(* IEC 61131-3 sources: F100R_S278_Temperville/MyController.device.xml.v3^/Plc Logic.plclogic.xml.v3^/Application.application.xml.v3^/10_EntradasSaidas, 3 files *)

(* ---- A_Principal_IO.prg.st ---- *)
PROGRAM A_Principal_IO

IF NOT xTesteEntradaSaidas THEN
	B_EspelhoEntradas();
	C_EspelhoSaida();
END_IF

(* ---- B_EspelhoEntradas.prg.st ---- *)
PROGRAM B_EspelhoEntradas
VAR

END_VAR

//TM262L10MESE8T - 0.1

ImgTesteEntradas[1]:=   xChCircuitoEmergenciaCC	:= xM0_1_DI0;//xChCircuitoEmergenciaCC
ImgTesteEntradas[2]:=   xChHabDesabCircuitoCC := xM0_1_DI1;//Reserva
ImgTesteEntradas[3]:=   xSaidaNobreakOk:= 	xM0_1_DI2;//xSaidaNobreakOk
ImgTesteEntradas[4]:=	xReleSeguranca:=	xM0_1_DI3;//xReleSeguranca

xInvVentilador01Habilitado:=true;//xM0_1_DI1;

//TM3XHSC202 - 0.2
ImgTesteEntradas[5]:=	xM0_2_DI0;// ENCODER
ImgTesteEntradas[6]:=	xM0_2_DI1;// ENCODER
ImgTesteEntradas[7]:=	xM0_2_DI2;// ENCODER
ImgTesteEntradas[8]:=	xM0_2_DI3;// ENCODER
ImgTesteEntradas[9]:=	xM0_2_DI4;// ENCODER
ImgTesteEntradas[10]:=	xM0_2_DI5;// ENCODER
ImgTesteEntradas[11]:=	xM0_2_DI6;// ENCODER
ImgTesteEntradas[12]:=	xM0_2_DI7;// ENCODER
ImgTesteEntradas[13]:=	xM0_2_DI8;// ENCODER
ImgTesteEntradas[14]:=	xM0_2_DI9;// ENCODER

//TM3XHSC202 - 0.3
ImgTesteEntradas[15]:=	xM0_3_DI0;// ENCODER
ImgTesteEntradas[16]:=	xM0_3_DI1;// ENCODER
ImgTesteEntradas[17]:=	xM0_3_DI2;// ENCODER
ImgTesteEntradas[18]:=	xM0_3_DI3;// ENCODER
ImgTesteEntradas[19]:=	xM0_3_DI4;// ENCODER
ImgTesteEntradas[20]:=	xM0_3_DI5;// ENCODER
ImgTesteEntradas[21]:=	xM0_3_DI6;// ENCODER
ImgTesteEntradas[22]:=	xM0_3_DI7;// ENCODER
ImgTesteEntradas[23]:=	xM0_3_DI8;// ENCODER
ImgTesteEntradas[24]:=	xM0_3_DI9;// ENCODER

//TM3DI32K - 0.4
ImgTesteEntradas[25]:= 	xChAvancaMesaEntrada	:= xM0_4_DI0;	//xChAvancaMesaEntrada
ImgTesteEntradas[26]:= 	xChRecuaMesaEntrada		:= xM0_4_DI1;	//xChRecuaMesaEntrada
ImgTesteEntradas[27]:= 	xSensorEntrada01		:= xM0_4_DI2;	//xSensorEntrada01
ImgTesteEntradas[28]:= 	xSensorEntrada02		:= xM0_4_DI3;	//xSensorEntrada02
ImgTesteEntradas[29]:= 	xSensorEntrada03		:= xM0_4_DI4;	//xSensorEntrada03
ImgTesteEntradas[30]:= 	xSensorEntrada04		:= xM0_4_DI5;	//xSensorEntrada04
ImgTesteEntradas[31]:= 	xSensorEntrada05		:= xM0_4_DI6;	//xSensorEntrada05
ImgTesteEntradas[32]:= 	xSensorEntrada06		:= xM0_4_DI7;  //xSensorEntrada06
ImgTesteEntradas[33]:= 	xSensorEntrada07		:= xM0_4_DI8;  //xSensorEntrada07
ImgTesteEntradas[34]:= 	xSensorEntrada08		:= xM0_4_DI9;  //xSensorEntrada08
ImgTesteEntradas[35]:= 	xBtGradeEntrada			:= xM0_4_DI10; //xBtGradeEntrada
ImgTesteEntradas[36]:= 	xBtHabilitaCarregamento	:= xM0_4_DI11; //xBtHabilitaCarregamento
ImgTesteEntradas[37]:= 	xBt02Emergencia			:= xM0_4_DI12; //xBt02Emergencia Mesa Entrada
ImgTesteEntradas[38]:= 	xSensorPortaEntrada		:= xM0_4_DI13; //xSensorPortaEntrada
ImgTesteEntradas[39]:= 	xSensorPortaSaida		:=	xM0_4_DI14; //xSensorPortaSaida
ImgTesteEntradas[40]:= 	xM0_4_DI15; //xSensorAbertoForno
ImgTesteEntradas[41]:=	xM0_4_DI16; //xSensorFechadoForno
ImgTesteEntradas[42]:=	xSensorAbertoResfriadorSup02:= xM0_4_DI17; //xSensorAbertoResfriadorSup02
ImgTesteEntradas[43]:=	xSensorFechadoResfriadorSup02:= xM0_4_DI18; //xSensorFechadoResfriadorSup02
ImgTesteEntradas[44]:=	xFcMaximoSegResfriadorSup02:= xM0_4_DI19; //xFcMaximoSegResfriadorSup02
ImgTesteEntradas[45]:=	xFcMinimoSegResfriadorSup02:= xM0_4_DI20; //xFcMinimoSegResfriadorSup02
ImgTesteEntradas[46]:=	xChAbreDuctosResfriadorSup02:= xM0_4_DI21; //xChAbreDuctosResfriadorSup02
ImgTesteEntradas[47]:=	xBt03Emergencia			:= xM0_4_DI22; //xBt03Emergencia Mesa Resfriador
ImgTesteEntradas[48]:=	xSensorDesligaMesaSaida	:= xM0_4_DI23; //xSensorDesligaMesaSaida
ImgTesteEntradas[49]:=	xSensorGradeSaidaUp		:= xM0_4_DI24; //xSensorGradeSaidaUp
ImgTesteEntradas[50]:=	xBtGradeSaida			:=	xM0_4_DI25;  //	xBtGradeSaida
ImgTesteEntradas[51]:=	xChAvancaMesaSaida		:= xM0_4_DI26; //xChAvancaMesaSaida
ImgTesteEntradas[52]:=	xChRecuaMesaSaida		:=	xM0_4_DI27; //xChRecuaMesaSaida
ImgTesteEntradas[53]:=	xBt04Emergencia			:= xM0_4_DI28; //xBt04Emergencia Mesa Saída
ImgTesteEntradas[54]:=	xSensorPositivoGuilhotina02:= xM0_4_DI29; //xSensorPositivoGuilhotina02
ImgTesteEntradas[55]:=	xSensorNegativoGuilhotina02:=xM0_4_DI30; //xSensorNegativoGuilhotina02
ImgTesteEntradas[56]:=	xSensorZeroGuilhotina02	:= xM0_4_DI31; //xSensorZeroGuilhotina02

//TM3DI32K - 3.1
ImgTesteEntradas[57]:= 	xChAutomaticoManual:= xM3_1_DI0;   //xChAutomaticoManual
ImgTesteEntradas[58]:= xBt01CalaAlarme:= xM3_1_DI1;   //xBt01CalaAlarme Mesa Controle
ImgTesteEntradas[59]:= xBt01Emergencia:= xM3_1_DI2;   //xBt01Emergencia Mesa Controle
ImgTesteEntradas[60]:= xPressaoBaixaMediaRede:= xM3_1_DI3;   //xPressaoBaixaMediaRede
ImgTesteEntradas[61]:= xPressaoMediaAltaRede:=	xM3_1_DI4;   //xPressaoMediaAltaRede
ImgTesteEntradas[62]:= xKaMotorOscilaResfr02Sup:= xM3_1_DI5;   //oscilantes
ImgTesteEntradas[63]:= xKaMotorOscilaResfr02Inf:= xM3_1_DI6;   //oscilantes
ImgTesteEntradas[64]:= xSensorOscilaResfr02Sup:= xM3_1_DI7;   //oscilantes
ImgTesteEntradas[65]:= xSensorOscilaResfr02Inf:= xM3_1_DI8;   //oscilantes
ImgTesteEntradas[66]:= xRetornoSsr01ConveccaoEnt:=	xM3_1_DI9;   //xRetornoSsr01ConveccaoEnt
ImgTesteEntradas[67]:= xRetornoSsr02ConveccaoEnt:=	xM3_1_DI10;  //xRetornoSsr02ConveccaoEnt
ImgTesteEntradas[68]:= xRetornoSsr03ConveccaoEnt:=	xM3_1_DI11;  //xRetornoSsr03ConveccaoEnt
ImgTesteEntradas[69]:= xRetornoSsrInferior[1]:= xM3_1_DI12;  //Retorno Circuito Resist Inf 01
ImgTesteEntradas[70]:= xRetornoSsrInferior[2]:= xM3_1_DI13;  //Retorno Circuito Resist Inf 02
ImgTesteEntradas[71]:= xRetornoSsrInferior[3]:= xM3_1_DI14;  //Retorno Circuito Resist Inf 03
ImgTesteEntradas[72]:= xRetornoSsrInferior[4]:= xM3_1_DI15;  //Retorno Circuito Resist Inf 04

//TM3DI32K - 3.2
ImgTesteEntradas[73]:= xRetornoSsrInferior[5]:= xM3_2_DI0;   //Retorno Circuito Resist Inf 05
ImgTesteEntradas[74]:= xRetornoSsrInferior[6]:= xM3_2_DI1;   //Retorno Circuito Resist Inf 06
ImgTesteEntradas[75]:= xRetornoSsrInferior[7]:= xM3_2_DI2;   //Retorno Circuito Resist Inf 07
ImgTesteEntradas[76]:= xRetornoSsrInferior[8]:= xM3_2_DI3;   //Retorno Circuito Resist Inf 08
ImgTesteEntradas[77]:= xRetornoSsrInferior[9]:= xM3_2_DI4;   //Retorno Circuito Resist Inf 09
ImgTesteEntradas[78]:= xRetornoSsrInferior[10]:= xM3_2_DI5;   //Retorno Circuito Resist Inf 10
ImgTesteEntradas[79]:= xRetornoSsrInferior[11]:= xM3_2_DI6;   //Retorno Circuito Resist Inf 11
ImgTesteEntradas[80]:= xRetornoSsrInferior[12]:= xM3_2_DI7;   //Retorno Circuito Resist Inf 12
ImgTesteEntradas[81]:= xRetornoSsrInferior[13]:= xM3_2_DI8;   //Retorno Circuito Resist Inf 13
ImgTesteEntradas[82]:= xRetornoSsrInferior[14]:= xM3_2_DI9;   //Retorno Circuito Resist Inf 14
ImgTesteEntradas[83]:= xRetornoSsrInferior[15]:= xM3_2_DI10;  //Retorno Circuito Resist Inf 15
ImgTesteEntradas[84]:= xRetornoSsrInferior[16]:= xM3_2_DI11;  //Retorno Circuito Resist Inf 16
ImgTesteEntradas[85]:= xRetornoSsrInferior[17]:= xM3_2_DI12;  //Retorno Circuito Resist Inf 17
ImgTesteEntradas[86]:= xRetornoSsrInferior[18]:= xM3_2_DI13;  //Retorno Circuito Resist Inf 18
ImgTesteEntradas[87]:= xRetornoSsrInferior[19]:= xM3_2_DI14;  //Retorno Circuito Resist Inf 19
ImgTesteEntradas[88]:= xRetornoSsrInferior[20]:= xM3_2_DI15;  //Retorno Circuito Resist Inf 20
ImgTesteEntradas[89]:= xRetornoSsrInferior[21]:= xM3_2_DI16;  //Retorno Circuito Resist Inf 21
ImgTesteEntradas[90]:= xRetornoSsrInferior[22]:= xM3_2_DI17;  //Retorno Circuito Resist Inf 22
ImgTesteEntradas[91]:= xRetornoSsrInferior[23]:= xM3_2_DI18;  //Retorno Circuito Resist Inf 23
ImgTesteEntradas[92]:= xRetornoSsrInferior[24]:= xM3_2_DI19;  //Retorno Circuito Resist Inf 24
ImgTesteEntradas[93]:= xRetornoSsrInferior[25]:= xM3_2_DI20;  //Retorno Circuito Resist Inf 25
ImgTesteEntradas[94]:= xRetornoSsrInferior[26]:= xM3_2_DI21;  //Retorno Circuito Resist Inf 26
ImgTesteEntradas[95]:= xRetornoSsrInferior[27]:= xM3_2_DI22;  //Retorno Circuito Resist Inf 27
ImgTesteEntradas[96]:= xRetornoSsrInferior[28]:= xM3_2_DI23;  //Retorno Circuito Resist Inf 28
ImgTesteEntradas[97]:= xRetornoSsrInferior[29]:= xM3_2_DI24;  //Retorno Circuito Resist Inf 29
ImgTesteEntradas[98]:= xRetornoSsrInferior[30]:= xM3_2_DI25;  //Retorno Circuito Resist Inf 30
ImgTesteEntradas[99]:= xRetornoSsrInferior[31]:= xM3_2_DI26;  //Retorno Circuito Resist Inf 31
ImgTesteEntradas[100]:= xRetornoSsrInferior[32]:= xM3_2_DI27;  //Retorno Circuito Resist Inf 32
ImgTesteEntradas[101]:=	xRetornoSsrInferior[33]:= xM3_2_DI28;  //Retorno Circuito Resist Inf 33
ImgTesteEntradas[102]:=	xRetornoSsrInferior[34]:= xM3_2_DI29;  //Retorno Circuito Resist Inf 34
ImgTesteEntradas[103]:=	xRetornoSsrInferior[35]:= xM3_2_DI30;  //Retorno Circuito Resist Inf 35
ImgTesteEntradas[104]:=	xRetornoSsrInferior[36]:= xM3_2_DI31;  //Retorno Circuito Resist Inf 36

//TM3DI32K - 4.1
ImgTesteEntradas[105]:=	xRetornoSsrInferior[37]:= xM4_1_DI0;   //Retorno Circuito Resist Inf 37
ImgTesteEntradas[106]:=	xRetornoSsrInferior[38]:= xM4_1_DI1;   //Retorno Circuito Resist Inf 38
ImgTesteEntradas[107]:=	xRetornoSsrInferior[39]:= xM4_1_DI2;   //Retorno Circuito Resist Inf 39
ImgTesteEntradas[108]:=	xRetornoSsrInferior[40]:= xM4_1_DI3;   //Retorno Circuito Resist Inf 40
ImgTesteEntradas[109]:=	xRetornoSsrInferior[41]:= xM4_1_DI4;   //Retorno Circuito Resist Inf 41
ImgTesteEntradas[110]:=	xRetornoSsrInferior[42]:= xM4_1_DI5;   //Retorno Circuito Resist Inf 42
ImgTesteEntradas[111]:=	xRetornoSsrInferior[43]:= xM4_1_DI6;   //Retorno Circuito Resist Inf 43
ImgTesteEntradas[112]:=	xRetornoSsrInferior[44]:= xM4_1_DI7;   //Retorno Circuito Resist Inf 44
ImgTesteEntradas[113]:=	xRetornoSsrInferior[45]:= xM4_1_DI8;   //Retorno Circuito Resist Inf 45
ImgTesteEntradas[114]:=	xRetornoSsrInferior[46]:= xM4_1_DI9;   //Retorno Circuito Resist Inf 46
ImgTesteEntradas[115]:=	xRetornoSsrInferior[47]:= xM4_1_DI10;  //Retorno Circuito Resist Inf 47
ImgTesteEntradas[116]:=	xRetornoSsrInferior[48]:= xM4_1_DI11;  //Retorno Circuito Resist Inf 48
ImgTesteEntradas[117]:=	xRetornoSsrInferior[49]:= xM4_1_DI12;  //Retorno Circuito Resist Inf 49
ImgTesteEntradas[118]:= xRetornoSsrInferior[50]:= xM4_1_DI13;  //Retorno Circuito Resist Inf 50
ImgTesteEntradas[119]:= xRetornoSsrSuperior[1]:= xM4_1_DI14;  //Retorno Circuito Resist Sup 01 - 51
ImgTesteEntradas[120]:= xRetornoSsrSuperior[2]:= xM4_1_DI15;  //Retorno Circuito Resist Sup 02 - 52
ImgTesteEntradas[121]:= xRetornoSsrSuperior[3]:= xM4_1_DI16;  //Retorno Circuito Resist Sup 03 - 53
ImgTesteEntradas[122]:= xRetornoSsrSuperior[4]:= xM4_1_DI17;  //Retorno Circuito Resist Sup 04 - 54
ImgTesteEntradas[123]:= xRetornoSsrSuperior[5]:= xM4_1_DI18;  //Retorno Circuito Resist Sup 05 - 55
ImgTesteEntradas[124]:= xRetornoSsrSuperior[6]:= xM4_1_DI19;  //Retorno Circuito Resist Sup 06 - 56
ImgTesteEntradas[125]:= xRetornoSsrSuperior[7]:= xM4_1_DI20;  //Retorno Circuito Resist Sup 07 - 57
ImgTesteEntradas[126]:= xRetornoSsrSuperior[8]:= xM4_1_DI21;  //Retorno Circuito Resist Sup 08 - 58
ImgTesteEntradas[127]:= xRetornoSsrSuperior[9]:= xM4_1_DI22;  //Retorno Circuito Resist Sup 09 - 59
ImgTesteEntradas[128]:= xRetornoSsrSuperior[10]:= xM4_1_DI23;  //Retorno Circuito Resist Sup 10 - 60
ImgTesteEntradas[129]:= xRetornoSsrSuperior[11]:= xM4_1_DI24;  //Retorno Circuito Resist Sup 11 - 61
ImgTesteEntradas[130]:= xRetornoSsrSuperior[12]:= xM4_1_DI25;  //Retorno Circuito Resist Sup 12 - 62
ImgTesteEntradas[131]:= xRetornoSsrSuperior[13]:= xM4_1_DI26;  //Retorno Circuito Resist Sup 13 - 63
ImgTesteEntradas[132]:= xRetornoSsrSuperior[14]:= xM4_1_DI27;  //Retorno Circuito Resist Sup 14 - 64
ImgTesteEntradas[133]:=	xRetornoSsrSuperior[15]:= xM4_1_DI28;  //Retorno Circuito Resist Sup 15 - 65
ImgTesteEntradas[134]:=	xRetornoSsrSuperior[16]:= xM4_1_DI29;  //Retorno Circuito Resist Sup 16 - 66
ImgTesteEntradas[135]:=	xRetornoSsrSuperior[17]:= xM4_1_DI30;  //Retorno Circuito Resist Sup 17 - 67
ImgTesteEntradas[136]:=	xRetornoSsrSuperior[18]:= xM4_1_DI31;  //Retorno Circuito Resist Sup 18 - 68

//TM3DI32K - 4.2
ImgTesteEntradas[137]:= xRetornoSsrSuperior[19]:= xM4_2_DI0;   //Retorno Circuito Resist Sup 19	- 69
ImgTesteEntradas[138]:= xRetornoSsrSuperior[20]:= xM4_2_DI1;   //Retorno Circuito Resist Sup 20	- 70
ImgTesteEntradas[139]:= xRetornoSsrSuperior[21]:= xM4_2_DI2;   //Retorno Circuito Resist Sup 21	- 71
ImgTesteEntradas[140]:= xRetornoSsrSuperior[22]:= xM4_2_DI3;   //Retorno Circuito Resist Sup 22	- 72
ImgTesteEntradas[141]:= xRetornoSsrSuperior[23]:= xM4_2_DI4;   //Retorno Circuito Resist Sup 23	- 73
ImgTesteEntradas[142]:= xRetornoSsrSuperior[24]:= xM4_2_DI5;   //Retorno Circuito Resist Sup 24	- 74
ImgTesteEntradas[143]:= xRetornoSsrSuperior[25]:= xM4_2_DI6;   //Retorno Circuito Resist Sup 25	- 75
ImgTesteEntradas[144]:= xRetornoSsrSuperior[26]:= xM4_2_DI7;   //Retorno Circuito Resist Sup 26	- 76
ImgTesteEntradas[145]:= xRetornoSsrSuperior[27]:= xM4_2_DI8;   //Retorno Circuito Resist Sup 27	- 77
ImgTesteEntradas[146]:= xRetornoSsrSuperior[28]:= xM4_2_DI9;   //Retorno Circuito Resist Sup 28 - 78
ImgTesteEntradas[147]:= xRetornoSsrSuperior[29]:= xM4_2_DI10;  //Retorno Circuito Resist Sup 29	- 79
ImgTesteEntradas[148]:= xRetornoSsrSuperior[30]:= xM4_2_DI11;  //Retorno Circuito Resist Sup 30	- 80
ImgTesteEntradas[149]:= xRetornoSsrSuperior[31]:= xM4_2_DI12;  //Retorno Circuito Resist Sup 31	- 81
ImgTesteEntradas[150]:= xRetornoSsrSuperior[32]:= xM4_2_DI13;  //Retorno Circuito Resist Sup 32	- 82
ImgTesteEntradas[151]:= xRetornoSsrSuperior[33]:= xM4_2_DI14;  //Retorno Circuito Resist Sup 33 - 83
ImgTesteEntradas[152]:= xRetornoSsrSuperior[34]:= xM4_2_DI15;  //Retorno Circuito Resist Sup 34 - 84
ImgTesteEntradas[153]:= xRetornoSsrSuperior[35]:= xM4_2_DI16;  //Retorno Circuito Resist Sup 35 - 85
ImgTesteEntradas[154]:= xRetornoSsrSuperior[36]:= xM4_2_DI17;  //Retorno Circuito Resist Sup 36 - 86
ImgTesteEntradas[155]:= xRetornoSsrSuperior[37]:= xM4_2_DI18;  //Retorno Circuito Resist Sup 37	- 87
ImgTesteEntradas[156]:= xRetornoSsrSuperior[38]:= xM4_2_DI19;  //Retorno Circuito Resist Sup 38	- 88
ImgTesteEntradas[157]:= xRetornoSsrSuperior[39]:= xM4_2_DI20;  //Retorno Circuito Resist Sup 39 - 89
ImgTesteEntradas[158]:= xRetornoSsrSuperior[40]:= xM4_2_DI21;  //Retorno Circuito Resist Sup 40	- 90
ImgTesteEntradas[159]:= xRetornoSsrSuperior[41]:= xM4_2_DI22;  //Retorno Circuito Resist Sup 41 - 91
ImgTesteEntradas[160]:= xRetornoSsrSuperior[42]:= xM4_2_DI23;  //Retorno Circuito Resist Sup 42 - 92
ImgTesteEntradas[161]:= xRetornoSsrSuperior[43]:= xM4_2_DI24;  //Retorno Circuito Resist Sup 43 - 93
ImgTesteEntradas[162]:= xRetornoSsrSuperior[44]:= xM4_2_DI25;  //Retorno Circuito Resist Sup 44 - 94
ImgTesteEntradas[163]:= xRetornoSsrSuperior[45]:= xM4_2_DI26;  //Retorno Circuito Resist Sup 45 - 95
ImgTesteEntradas[164]:= xRetornoSsrSuperior[46]:= xM4_2_DI27;  //Retorno Circuito Resist Sup 46 - 96
ImgTesteEntradas[165]:=	xRetornoSsrSuperior[47]:= xM4_2_DI28;  //Retorno Circuito Resist Sup 47 - 97
ImgTesteEntradas[166]:=	xRetornoSsrSuperior[48]:= xM4_2_DI29;  //Retorno Circuito Resist Sup 48 - 98
ImgTesteEntradas[167]:=	xRetornoSsrSuperior[49]:= xM4_2_DI30;  //Retorno Circuito Resist Sup 49 - 99
ImgTesteEntradas[168]:=	xRetornoSsrSuperior[50]:= xM4_2_DI31;  //Retorno Circuito Resist Sup 50 - 100

ImgEncoder[1]:=dValorEncoderForno;
ImgEncoder[2]:=dValorEncoderResfriador;
ImgEncoder[3]:=dValorEncoderDuctosResfriadorSup01;
ImgEncoder[4]:=dValorEncoderDuctosResfriadorInf01;
ImgEncoder[5]:=dValorEncoderDuctosResfriadorSup02;
ImgEncoder[6]:=dValorEncoderDuctosResfriadorInf02;
ImgEncoder[7]:=dValorEncoderGuilhotinaResfriador01;
ImgEncoder[8]:=dValorEncoderGuilhotinaResfriador02;

(* ---- C_EspelhoSaida.prg.st ---- *)
PROGRAM C_EspelhoSaida
VAR

END_VAR

//TM262L10MESE8T - 0.1
xM0_1_DQ0:=TRUE ;// ByPass
xM0_1_DQ1:=xSinalLumVerm; //Vermelho
xM0_1_DQ2:=xSinalLumAmar; //Amarelo
xM0_1_DQ3:=xSinalLumVerd; //Verde

//TM3XHSC202 - 0.2
xM0_2_DQ0:=xVentiladoresPainel;
xM0_2_DQ1:=xVentiladoresSsr;
xM0_2_DQ2:=xValvulaGradeEntrada;
xM0_2_DQ3:=xValvPortaEntradaForno;
xM0_2_DQ4:=xValvPortaSaidaForno;
xM0_2_DQ5:=xValvulaGradeSaida;
xM0_2_DQ6:=xValvulaDamperDifusor;
xM0_2_DQ7:=xLedCargaForno;

//TM3XHSC202 - 0.3
xM0_3_DQ0:=NOT xReleSeguranca;
xM0_3_DQ1:=xAlarmeSonoro;
xM0_3_DQ2:=xMotorOscilaResfr02Sup;// oscila sup
xM0_3_DQ3:=xMotorOscilaResfr02Inf;// oscila inf
xM0_3_DQ4:=FALSE;// RESERVA
xM0_3_DQ5:=FALSE;// RESERVA
xM0_3_DQ6:=FALSE;// RESERVA
xM0_3_DQ7:=FALSE;// RESERVA

//TM3DM24K - 3.1
xM3_1_DQ0:= FALSE;// RESERVA
xM3_1_DQ1:= FALSE;// RESERVA
xM3_1_DQ2:= FALSE;// RESERVA
xM3_1_DQ3:= xReleSsrConveccaoEnt;
xM3_1_DQ4:= xReleSsrInferior[1] OR xSaidaReleRampaPatamarInf[1];
xM3_1_DQ5:= xReleSsrInferior[2] OR xSaidaReleRampaPatamarInf[2];
xM3_1_DQ6:= xReleSsrInferior[3] OR xSaidaReleRampaPatamarInf[3];
xM3_1_DQ7:= xReleSsrInferior[4] OR xSaidaReleRampaPatamarInf[4];

//TM3DQ32TK - 3.3
xM3_3_DQ0:= xReleSsrInferior[5] OR xSaidaReleRampaPatamarInf[5]; // xReleSsrInferior[5]
xM3_3_DQ1:= xReleSsrInferior[6] OR xSaidaReleRampaPatamarInf[6]; // xReleSsrInferior[6]
xM3_3_DQ2:= xReleSsrInferior[7] OR xSaidaReleRampaPatamarInf[7]; // xReleSsrInferior[7]
xM3_3_DQ3:= xReleSsrInferior[8] OR xSaidaReleRampaPatamarInf[8]; // xReleSsrInferior[8]
xM3_3_DQ4:= xReleSsrInferior[9] OR xSaidaReleRampaPatamarInf[9]; // xReleSsrInferior[9]
xM3_3_DQ5:= xReleSsrInferior[10] OR xSaidaReleRampaPatamarInf[10];// xReleSsrInferior[10]
xM3_3_DQ6:= xReleSsrInferior[11] OR xSaidaReleRampaPatamarInf[11];// xReleSsrInferior[11]
xM3_3_DQ7:= xReleSsrInferior[12] OR xSaidaReleRampaPatamarInf[12];// xReleSsrInferior[12]
xM3_3_DQ8:= xReleSsrInferior[13] OR xSaidaReleRampaPatamarInf[13];// xReleSsrInferior[13]
xM3_3_DQ9:= xReleSsrInferior[14] OR xSaidaReleRampaPatamarInf[14];// xReleSsrInferior[14]
xM3_3_DQ10:=xReleSsrInferior[15] OR xSaidaReleRampaPatamarInf[15];// xReleSsrInferior[15]
xM3_3_DQ11:=xReleSsrInferior[16] OR xSaidaReleRampaPatamarInf[16];// xReleSsrInferior[16]
xM3_3_DQ12:=xReleSsrInferior[17] OR xSaidaReleRampaPatamarInf[17];// xReleSsrInferior[17]
xM3_3_DQ13:=xReleSsrInferior[18] OR xSaidaReleRampaPatamarInf[18];// xReleSsrInferior[18]
xM3_3_DQ14:=xReleSsrInferior[19] OR xSaidaReleRampaPatamarInf[19];// xReleSsrInferior[19]
xM3_3_DQ15:=xReleSsrInferior[20] OR xSaidaReleRampaPatamarInf[20];// xReleSsrInferior[20]
xM3_3_DQ16:=xReleSsrInferior[21] OR xSaidaReleRampaPatamarInf[21];// xReleSsrInferior[21]
xM3_3_DQ17:=xReleSsrInferior[22] OR xSaidaReleRampaPatamarInf[22];// xReleSsrInferior[22]
xM3_3_DQ18:=xReleSsrInferior[23] OR xSaidaReleRampaPatamarInf[23];// xReleSsrInferior[23]
xM3_3_DQ19:=xReleSsrInferior[24] OR xSaidaReleRampaPatamarInf[24];// xReleSsrInferior[24]
xM3_3_DQ20:=xReleSsrInferior[25] OR xSaidaReleRampaPatamarInf[25];// xReleSsrInferior[25]
xM3_3_DQ21:=xReleSsrInferior[26] OR xSaidaReleRampaPatamarInf[26];// xReleSsrInferior[26]
xM3_3_DQ22:=xReleSsrInferior[27] OR xSaidaReleRampaPatamarInf[27];// xReleSsrInferior[27]
xM3_3_DQ23:=xReleSsrInferior[28] OR xSaidaReleRampaPatamarInf[28];// xReleSsrInferior[28]
xM3_3_DQ24:=xReleSsrInferior[29] OR xSaidaReleRampaPatamarInf[29];// xReleSsrInferior[29]
xM3_3_DQ25:=xReleSsrInferior[30] OR xSaidaReleRampaPatamarInf[30];// xReleSsrInferior[30]
xM3_3_DQ26:=xReleSsrInferior[31] OR xSaidaReleRampaPatamarInf[31];// xReleSsrInferior[31]
xM3_3_DQ27:=xReleSsrInferior[32] OR xSaidaReleRampaPatamarInf[32];// xReleSsrInferior[32]
xM3_3_DQ28:=xReleSsrInferior[33] OR xSaidaReleRampaPatamarInf[33];// xReleSsrInferior[33]
xM3_3_DQ29:=xReleSsrInferior[34] OR xSaidaReleRampaPatamarInf[34];// xReleSsrInferior[34]
xM3_3_DQ30:=xReleSsrInferior[35] OR xSaidaReleRampaPatamarInf[35];// xReleSsrInferior[35]
xM3_3_DQ31:=xReleSsrInferior[36] OR xSaidaReleRampaPatamarInf[36];// xReleSsrInferior[36]

//TM3DQ32TK - 4.3
xM4_3_DQ0:= xReleSsrInferior[37] OR xSaidaReleRampaPatamarInf[37]; // xReleSsrInferior[37]
xM4_3_DQ1:= xReleSsrInferior[38] OR xSaidaReleRampaPatamarInf[38]; // xReleSsrInferior[38]
xM4_3_DQ2:= xReleSsrInferior[39] OR xSaidaReleRampaPatamarInf[39]; // xReleSsrInferior[39]
xM4_3_DQ3:= xReleSsrInferior[40] OR xSaidaReleRampaPatamarInf[40]; // xReleSsrInferior[40]
xM4_3_DQ4:= xReleSsrInferior[41] OR xSaidaReleRampaPatamarInf[41]; // xReleSsrInferior[41]
xM4_3_DQ5:= xReleSsrInferior[42] OR xSaidaReleRampaPatamarInf[42]; // xReleSsrInferior[42]
xM4_3_DQ6:= xReleSsrInferior[43] OR xSaidaReleRampaPatamarInf[43]; // xReleSsrInferior[43]
xM4_3_DQ7:= xReleSsrInferior[44] OR xSaidaReleRampaPatamarInf[44]; // xReleSsrInferior[44]
xM4_3_DQ8:= xReleSsrInferior[45] OR xSaidaReleRampaPatamarInf[45]; // xReleSsrInferior[45]
xM4_3_DQ9:= xReleSsrInferior[46] OR xSaidaReleRampaPatamarInf[46]; // xReleSsrInferior[46]
xM4_3_DQ10:=xReleSsrInferior[47] OR xSaidaReleRampaPatamarInf[47]; // xReleSsrInferior[47]
xM4_3_DQ11:=xReleSsrInferior[48] OR xSaidaReleRampaPatamarInf[48]; // xReleSsrInferior[48]
xM4_3_DQ12:=xReleSsrInferior[49] OR xSaidaReleRampaPatamarInf[49]; // xReleSsrInferior[49]
xM4_3_DQ13:=xReleSsrInferior[50] OR xSaidaReleRampaPatamarInf[50]; // xReleSsrInferior[50]
xM4_3_DQ14:=xReleSsrSuperior[1] OR xSaidaReleRampaPatamarSup[1]; // xReleSsrSuperior[1] - 51
xM4_3_DQ15:=xReleSsrSuperior[2] OR xSaidaReleRampaPatamarSup[2]; // xReleSsrSuperior[2] - 52
xM4_3_DQ16:=xReleSsrSuperior[3] OR xSaidaReleRampaPatamarSup[3]; // xReleSsrSuperior[3] - 53
xM4_3_DQ17:=xReleSsrSuperior[4] OR xSaidaReleRampaPatamarSup[4]; // xReleSsrSuperior[4] - 54
xM4_3_DQ18:=xReleSsrSuperior[5] OR xSaidaReleRampaPatamarSup[5]; // xReleSsrSuperior[5] - 55
xM4_3_DQ19:=xReleSsrSuperior[6] OR xSaidaReleRampaPatamarSup[6]; // xReleSsrSuperior[6] - 56
xM4_3_DQ20:=xReleSsrSuperior[7] OR xSaidaReleRampaPatamarSup[7]; // xReleSsrSuperior[7] - 57
xM4_3_DQ21:=xReleSsrSuperior[8] OR xSaidaReleRampaPatamarSup[8]; // xReleSsrSuperior[8] - 58
xM4_3_DQ22:=xReleSsrSuperior[9] OR xSaidaReleRampaPatamarSup[9]; // xReleSsrSuperior[9] - 59
xM4_3_DQ23:=xReleSsrSuperior[10] OR xSaidaReleRampaPatamarSup[10]; // xReleSsrSuperior[10] - 60
xM4_3_DQ24:=xReleSsrSuperior[11] OR xSaidaReleRampaPatamarSup[11]; // xReleSsrSuperior[11] - 61
xM4_3_DQ25:=xReleSsrSuperior[12] OR xSaidaReleRampaPatamarSup[12]; // xReleSsrSuperior[12] - 62
xM4_3_DQ26:=xReleSsrSuperior[13] OR xSaidaReleRampaPatamarSup[13]; // xReleSsrSuperior[13] - 63
xM4_3_DQ27:=xReleSsrSuperior[14] OR xSaidaReleRampaPatamarSup[14]; // xReleSsrSuperior[14] - 64
xM4_3_DQ28:=xReleSsrSuperior[15] OR xSaidaReleRampaPatamarSup[15]; // xReleSsrSuperior[15] - 65
xM4_3_DQ29:=xReleSsrSuperior[16] OR xSaidaReleRampaPatamarSup[16]; // xReleSsrSuperior[16] - 66
xM4_3_DQ30:=xReleSsrSuperior[17] OR xSaidaReleRampaPatamarSup[17]; // xReleSsrSuperior[17] - 67
xM4_3_DQ31:=xReleSsrSuperior[18] OR xSaidaReleRampaPatamarSup[18]; // xReleSsrSuperior[18] - 68

//TM3DQ32TK - 4.4
xM4_4_DQ0:= xReleSsrSuperior[19] OR xSaidaReleRampaPatamarSup[19]; // xReleSsrSuperior[19] - 69
xM4_4_DQ1:= xReleSsrSuperior[20] OR xSaidaReleRampaPatamarSup[20]; // xReleSsrSuperior[20] - 70
xM4_4_DQ2:= xReleSsrSuperior[21] OR xSaidaReleRampaPatamarSup[21]; // xReleSsrSuperior[21] - 71
xM4_4_DQ3:= xReleSsrSuperior[22] OR xSaidaReleRampaPatamarSup[22]; // xReleSsrSuperior[22] - 72
xM4_4_DQ4:= xReleSsrSuperior[23] OR xSaidaReleRampaPatamarSup[23]; // xReleSsrSuperior[23] - 73
xM4_4_DQ5:= xReleSsrSuperior[24] OR xSaidaReleRampaPatamarSup[24]; // xReleSsrSuperior[24] - 74
xM4_4_DQ6:= xReleSsrSuperior[25] OR xSaidaReleRampaPatamarSup[25]; // xReleSsrSuperior[25] - 75
xM4_4_DQ7:= xReleSsrSuperior[26] OR xSaidaReleRampaPatamarSup[26]; // xReleSsrSuperior[26] - 76
xM4_4_DQ8:= xReleSsrSuperior[27] OR xSaidaReleRampaPatamarSup[27]; // xReleSsrSuperior[27] - 77
xM4_4_DQ9:= xReleSsrSuperior[28] OR xSaidaReleRampaPatamarSup[28]; // xReleSsrSuperior[28] - 78
xM4_4_DQ10:=xReleSsrSuperior[29] OR xSaidaReleRampaPatamarSup[29]; // xReleSsrSuperior[29] - 79
xM4_4_DQ11:=xReleSsrSuperior[30] OR xSaidaReleRampaPatamarSup[30]; // xReleSsrSuperior[30] - 80
xM4_4_DQ12:=xReleSsrSuperior[31] OR xSaidaReleRampaPatamarSup[31]; // xReleSsrSuperior[31] - 81
xM4_4_DQ13:=xReleSsrSuperior[32] OR xSaidaReleRampaPatamarSup[32]; // xReleSsrSuperior[32] - 82
xM4_4_DQ14:=xReleSsrSuperior[33] OR xSaidaReleRampaPatamarSup[33]; // xReleSsrSuperior[33] - 83
xM4_4_DQ15:=xReleSsrSuperior[34] OR xSaidaReleRampaPatamarSup[34]; // xReleSsrSuperior[34] - 84
xM4_4_DQ16:=xReleSsrSuperior[35] OR xSaidaReleRampaPatamarSup[35]; // xReleSsrSuperior[35] - 85
xM4_4_DQ17:=xReleSsrSuperior[36] OR xSaidaReleRampaPatamarSup[36]; // xReleSsrSuperior[36] - 86
xM4_4_DQ18:=xReleSsrSuperior[37] OR xSaidaReleRampaPatamarSup[37]; // xReleSsrSuperior[37] - 87
xM4_4_DQ19:=xReleSsrSuperior[38] OR xSaidaReleRampaPatamarSup[38]; // xReleSsrSuperior[38] - 88
xM4_4_DQ20:=xReleSsrSuperior[39] OR xSaidaReleRampaPatamarSup[39]; // xReleSsrSuperior[39] - 89
xM4_4_DQ21:=xReleSsrSuperior[40] OR xSaidaReleRampaPatamarSup[40]; // xReleSsrSuperior[40] - 90
xM4_4_DQ22:=xReleSsrSuperior[41] OR xSaidaReleRampaPatamarSup[41]; // xReleSsrSuperior[41] - 91
xM4_4_DQ23:=xReleSsrSuperior[42] OR xSaidaReleRampaPatamarSup[42]; // xReleSsrSuperior[42] - 92
xM4_4_DQ24:=xReleSsrSuperior[43] OR xSaidaReleRampaPatamarSup[43]; // xReleSsrSuperior[43] - 93
xM4_4_DQ25:=xReleSsrSuperior[44] OR xSaidaReleRampaPatamarSup[44]; // xReleSsrSuperior[44] - 94
xM4_4_DQ26:=xReleSsrSuperior[45] OR xSaidaReleRampaPatamarSup[45]; // xReleSsrSuperior[45] - 95
xM4_4_DQ27:=xReleSsrSuperior[46] OR xSaidaReleRampaPatamarSup[46]; // xReleSsrSuperior[46] - 96
xM4_4_DQ28:=xReleSsrSuperior[47] OR xSaidaReleRampaPatamarSup[47]; // xReleSsrSuperior[47] - 97
xM4_4_DQ29:=xReleSsrSuperior[48] OR xSaidaReleRampaPatamarSup[48]; // xReleSsrSuperior[48] - 98
xM4_4_DQ30:=xReleSsrSuperior[49] OR xSaidaReleRampaPatamarSup[49]; // xReleSsrSuperior[49] - 99
xM4_4_DQ31:=xReleSsrSuperior[50] OR xSaidaReleRampaPatamarSup[50]; // xReleSsrSuperior[50] - 100
